FUNCTION_BLOCK PendingRequestGenerator
  (* Standard: 61499-2 *)
  (* Version 0.1, 2014-00-16, Canto-Air, CANTO-AIR-PC *)
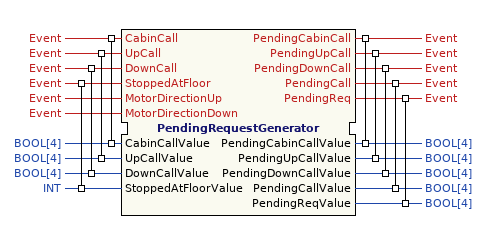
  EVENT_INPUT
    CabinCall WITH CabinCallValue;
    UpCall WITH UpCallValue;
    DownCall WITH DownCallValue;
    StoppedAtFloor WITH StoppedAtFloorValue;
    MotorDirectionUp;
    MotorDirectionDown;
  END_EVENT
  EVENT_OUTPUT
    PendingCabinCall WITH PendingCabinCallValue;
    PendingUpCall WITH PendingUpCallValue;
    PendingDownCall WITH PendingDownCallValue;
    PendingCall WITH PendingCallValue;
    PendingReq WITH PendingReqValue;
  END_EVENT
  VAR_INPUT
    CabinCallValue : ARRAY [0..3] OF BOOL;
    UpCallValue : ARRAY [0..3] OF BOOL;
    DownCallValue : ARRAY [0..3] OF BOOL;
    StoppedAtFloorValue : INT;
  END_VAR
  VAR_OUTPUT
    PendingCabinCallValue : ARRAY [0..3] OF BOOL;
    PendingUpCallValue : ARRAY [0..3] OF BOOL;
    PendingDownCallValue : ARRAY [0..3] OF BOOL;
    PendingCallValue : ARRAY [0..3] OF BOOL;
    PendingReqValue : ARRAY [0..3] OF BOOL;
  END_VAR
  VAR
    preCallRequest : BOOL;
    preMotorDirectionDown : BOOL;
    preMotorDirectionUp : BOOL;
  END_VAR
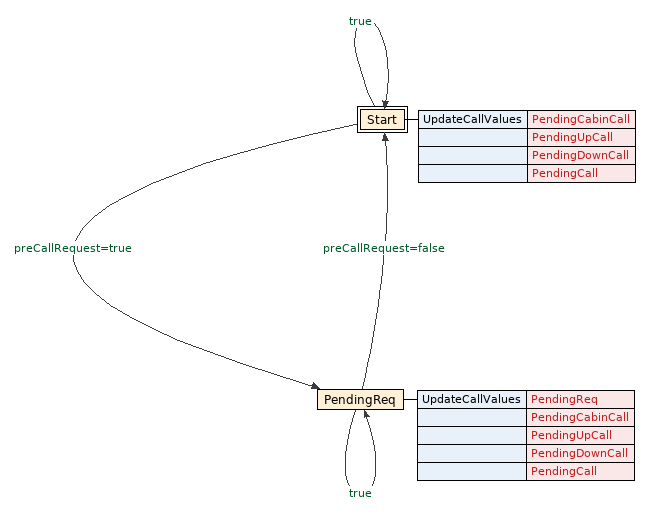
  EC_STATES
    Start : UpdateCallValues -> PendingCabinCall, -> PendingUpCall, -> PendingDownCall, -> PendingCall;
    PendingReq : UpdateCallValues -> PendingReq, -> PendingCabinCall, -> PendingUpCall, -> PendingDownCall, -> PendingCall;
  END_STATES
  EC_TRANSITIONS
    Start TO PendingReq := preCallRequest=true;
    Start TO Start := true;
    PendingReq TO Start := preCallRequest=false;
    PendingReq TO PendingReq := true;
  END_TRANSITIONS
  ALGORITHM UpdateCallValues IN C:
int i = 0;
//update PendingCabinCall
if (me->_input.event.CabinCall) {
	for (i = 0; i < 4; ++i) {
		me->PendingCabinCallValue[i] |= me->CabinCallValue[i];
	}
}
if (me->_input.event.StoppedAtFloor) {
	me->PendingCabinCallValue[me->StoppedAtFloorValue] = 0;
}
//update PendingUpCall
int hasUpRequests = 0;
if (me->_input.event.UpCall) {
	for (i = 0; i < 4; ++i) {
		me->PendingUpCallValue[i] |= me->UpCallValue[i];
		hasUpRequests|= me->UpCallValue[i];
	}
}
//update PendingDownCall
int hasDownRequests = 0;
if (me->_input.event.DownCall) {
	for (i = 0; i < 4; ++i) {
		me->PendingDownCallValue[i] |= me->DownCallValue[i];
		hasDownRequests |= me->DownCallValue[i];
	}
}
if ((me->_input.event.StoppedAtFloor&&me->preMotorDirectionUp) || (hasDownRequests==0)) {
	me->PendingUpCallValue[me->StoppedAtFloorValue] = 0;
}
if ((me->_input.event.StoppedAtFloor&&me->preMotorDirectionDown) || (hasUpRequests==0)) {
	me->PendingDownCallValue[me->StoppedAtFloorValue] = 0;
}
me->preCallRequest = 0;
//update PendingCall
for (i = 0; i < 4; ++i) {
    me->PendingCallValue[i] |=  me->PendingCabinCallValue[i] ||  me->PendingUpCallValue[i] || me->PendingDownCallValue[i];
	me->preCallRequest |= me->PendingCallValue[i];
}
if (me->_input.event.StoppedAtFloor) {
	me->PendingCallValue[me->StoppedAtFloorValue] = 0;
}
//update PendingReq
for (i = 0; i < 4; ++i) {
    me->PendingReqValue[i] = me->PendingCallValue[i];
}
me->preMotorDirectionUp = me->_input.event.MotorDirectionUp;
me->preMotorDirectionDown = me->_input.event.MotorDirectionDown;
  END_ALGORITHM
END_FUNCTION_BLOCK
